TYPE EM_Machine_SIM :
STRUCT
END_STRUCT
END_TYPE

(* stored: Version 1.1.0.1, ProductVersion 3.1.4024.12
   DUT EM_Machine_SIM: Id {67fea55f-f507-4f6d-99a1-4c8328caf8ed} *)
